// TIA Portal V17 export
// export: Created 2024-08-20T10:59:42.1994753Z, ExportSetting WithDefaults, DisplayName Totally Integrated Automation Portal, DisplayVersion V17 Update 4, DisplayName TIA Portal Openness, DisplayVersion V17 Update 4, DisplayName TIA Portal Version Control Interface, DisplayVersion V17, DisplayName STEP 7 Professional, DisplayVersion V17 Update 4, DisplayName STEP 7 Safety, DisplayVersion V17, DisplayName WinCC Advanced, DisplayVersion V17 Update 4
DATA_BLOCK "Digitais"   // DB300
{ S7_Optimized_Access := 'FALSE' }
VERSION : 0.1
// stored: AutoNumber false, DBAccessibleFromOPCUA true, IsOnlyStoredInLoadMemory false, IsWriteProtectedInAS false
   VAR RETAIN
      "MB-01-YSH" : Bool;   // Elevatoria principal 1 ligado
      "MB-01-YR" : Bool;   // Elevatoria principal 1 remoto
      "MB-01-YF" : Bool;   // Elevatoria principal 1 falha
      "MB-01-YFF" : Bool;   // Elevatoria principal 1 falta de fase
      "MB-01-MM" : Bool;   // Elevatoria principal 1 modo manutenção
      "MB-01-MA" : Bool;   // Elevatoria principal 1 modo automatico
      "MB-01-EMER" : Bool;   // Elevatoria principal 1 emergencia
      "MB-01-MN" : Bool;   // Elevatoria principal 1 modo normal
      "MB-01-ML" : Bool;   // Elevatoria principal 1 modo local
      "MB-01-YFI" : Bool;   // Elevatoria principal 1 com falha no inversor
      "MB-01-YFA" : Bool;   // Elevatoria principal 1 com falha no acionamento
      "MB-01-YPTA" : Bool;   // Elevatoria principal 1 com proteção térmica atuada
      "MB-01-HM" : Bool;   // Elevatoria principal 1 habilita manutenção
      "MB-01-RST" : Bool;   // Elevatoria principal 1 reset
      "MB-01-INTRU" : Bool;   // Elevatoria principal 1 intrusão no painel
      "MB-01-YFB" : Bool;   // Elevatoria principal 1 defeito na bomba
      "MB-02-YSH" : Bool;   // Elevatoria principal 2 ligado
      "MB-02-YR" : Bool;   // Elevatoria principal 2 remoto
      "MB-02-YF" : Bool;   // Elevatoria principal 2 falha
      "MB-02-YFF" : Bool;   // Elevatoria principal 2 falta de fase
      "MB-02-MM" : Bool;   // Elevatoria principal 2 modo manutenção
      "MB-02-MA" : Bool;   // Elevatoria principal 2 modo automatico
      "MB-02-EMER" : Bool;   // Elevatoria principal 2 emergencia
      "MB-02-MN" : Bool;   // Elevatoria principal 2 modo normal
      "MB-02-ML" : Bool;   // Elevatoria principal 2 modo local
      "MB-02-YFI" : Bool;   // Elevatoria principal 2 com falha no inversor
      "MB-02-YFA" : Bool;   // Elevatoria principal 2 com falha no acionamento
      "MB-02-YPTA" : Bool;   // Elevatoria principal 2 com proteção térmica atuada
      "MB-02-HM" : Bool;   // Elevatoria principal 2 habilita manutenção
      "MB-02-RST" : Bool;   // Elevatoria principal 2 reset
      "MB-02-INTRU" : Bool;   // Elevatoria principal 2 intrusão no painel
      "MB-02-YFB" : Bool;   // Elevatoria principal 2 defeito na bomba
      "MB-03-YSH" : Bool;   // Elevatoria principal 3 ligado
      "MB-03-YR" : Bool;   // Elevatoria principal 3 remoto
      "MB-03-YF" : Bool;   // Elevatoria principal 3 falha
      "MB-03-YFF" : Bool;   // Elevatoria principal 3 falta de fase
      "MB-03-MM" : Bool;   // Elevatoria principal 3 modo manutenção
      "MB-03-MA" : Bool;   // Elevatoria principal 3 modo automatico
      "MB-03-EMER" : Bool;   // Elevatoria principal 3 emergencia
      "MB-03-MN" : Bool;   // Elevatoria principal 3 modo normal
      "MB-03-ML" : Bool;   // Elevatoria principal 3 modo local
      "MB-03-YFI" : Bool;   // Elevatoria principal 3 com falha no inversor
      "MB-03-YFA" : Bool;   // Elevatoria principal 3 com falha no acionamento
      "MB-03-YPTA" : Bool;   // Elevatoria principal 3 com proteção térmica atuada
      "MB-03-HM" : Bool;   // Elevatoria principal 3 habilita manutenção
      "MB-03-RST" : Bool;   // Elevatoria principal 3 reset
      "MB-03-INTRU" : Bool;   // Elevatoria principal 3 intrusão no painel
      "MB-03-YFB" : Bool;   // Elevatoria principal 3 defeito na bomba
      "MB-04-YSH" : Bool;   // Elevatoria principal 4 ligado
      "MB-04-YR" : Bool;   // Elevatoria principal 4 remoto
      "MB-04-YF" : Bool;   // Elevatoria principal 4 falha
      "MB-04-YFF" : Bool;   // Elevatoria principal 4 falta de fase
      "MB-04-MM" : Bool;   // Elevatoria principal 4 modo manutenção
      "MB-04-MA" : Bool;   // Elevatoria principal 4 modo automatico
      "MB-04-EMER" : Bool;   // Elevatoria principal 4 emergencia
      "MB-04-MN" : Bool;   // Elevatoria principal 4 modo normal
      "MB-04-ML" : Bool;   // Elevatoria principal 4 modo local
      "MB-04-YFI" : Bool;   // Elevatoria principal 4 com falha no inversor
      "MB-04-YFA" : Bool;   // Elevatoria principal 4 com falha no acionamento
      "MB-04-YPTA" : Bool;   // Elevatoria principal 4 com proteção térmica atuada
      "MB-04-HM" : Bool;   // Elevatoria principal 4 habilita manutenção
      "MB-04-RST" : Bool;   // Elevatoria principal 4 reset
      "MB-04-INTRU" : Bool;   // Elevatoria principal 4 intrusão no painel
      "MB-04-YFB" : Bool;   // Elevatoria principal 4 defeito na bomba
      "LIT_001-AL8" : Bool;   // Disponível para alarme
      "LIT_001-AL9" : Bool;   // Disponível para alarme
      "LIT_001-AL10" : Bool;   // Disponível para alarme
      "LIT_001-AL11" : Bool;   // Disponível para alarme
      "LIT_001-AL12" : Bool;   // Disponível para alarme
      "LIT_001-AL13" : Bool;   // Disponível para alarme
      "LIT_001-AL14" : Bool;   // Disponível para alarme
      "LIT_001-AL15" : Bool;   // Disponível para alarme
      "LIT_001-YHH" : Bool;   // Alarme de nível muito alto do tanque
      "LIT_001-YH" : Bool;   // Alarme de nível alto do tanque
      "LIT_001-YL" : Bool;   // Alarme de nível baixo do tanque
      "LIT_001-YLL" : Bool;   // Alarme de nível muito baixo do tanque
      "LIT_001-YFS" : Bool;   // Transmissor de nível do tanque com falha de sinal
      "LIT_001-AL5" : Bool;   // Disponível para alarme
      "LIT_001-AL6" : Bool;   // Disponível para alarme
      "LIT_001-AL7" : Bool;   // Disponível para alarme
      PCM_EEE_EMER : Bool;   // PCM-E-CF-01-04 BOTAO DE EMERGENCIA - ATUADO
      PCM_EEE_K27 : Bool;   // PCM-E-CF-01-04 RELE DE PROTECAO FUNCAO 27 - ATUADO
      PCM_EEE_DISJ_LIG : Bool;   // PCM-E-CF-01-04 DISJUNTOR GERAL STATUS - LIGADO
      PCM_EEE_DISJ_DESLIG : Bool;   // PCM-E-CF-01-04 DISJUNTOR GERAL STATUS - DESLIGADO
      PCM_EEE_DISJ_YFAL : Bool;   // PCM-E-CF-01-04 DISJUNTOR GERAL STATUS - FALHA
      PCM_EEE_DISJ_FAL_GR : Bool;   // PCM-E-CF-01-04 FALHA GERAL ATUADO
      PCM_EEE_TR01_KA3 : Bool;   // PCM-E-CF-01-04 TRANSFORMADOR -TR-01 ALARME TEMP 150°
      PCM_EEE_TR01_KA4 : Bool;   // PCM-E-CF-01-04 TRANSFORMADOR -TR-01 ALARME TEMP 155°
      PCM_EEE_TR01_KA5 : Bool;   // PCM-E-CF-01-04 TRANSFORMADOR -TR-01 FALHA PROTECAO
      PCM_EEE_INTRU : Bool;   // PCM-E-CF-01-04 INTRUSAO NO PAINEL (COLUNA 01~04)
      PCM_EEE_RSERVA_0 : Bool;   // PCM-E-CF-01-04 BIT RESERVA DA WORD
      PCM_EEE_RSERVA_1 : Bool;   // PCM-E-CF-01-04 BIT RESERVA DA WORD
      PCM_EEE_RSERVA_2 : Bool;   // PCM-E-CF-01-04 BIT RESERVA DA WORD
      PCM_EEE_RSERVA_3 : Bool;   // PCM-E-CF-01-04 BIT RESERVA DA WORD
      PCM_EEE_RSERVA_4 : Bool;   // PCM-E-CF-01-04 BIT RESERVA DA WORD
      PCM_EEE_RSERVA_5 : Bool;   // PCM-E-CF-01-04 BIT RESERVA DA WORD
      QGBT_EMER : Bool;   // QGBT-AUX-01 BOTAO DE EMERGENCIA ATUADO
      QGBT_K27 : Bool;   // QGBT-AUX-01 RELE DE PROTECAO FUNCAO 27/59 ATUADO
      QGBT_DJL : Bool;   // QGBT-AUX-01 DISJUNTOR GERAL STATUS - LIGADO
      QGBT_DJD : Bool;   // QGBT-AUX-01 DISJUNTOR GERAL STATUS - DESLIGADO
      QGBT_DJYFAL : Bool;   // QGBT-AUX-01 DISJUNTOR GERAL FALHA - TRIP
      QGBT_INTRU : Bool;   // QGBT-AUX-01 INTRUSAO NO PAINEL
      QGBT_RESERVA_0 : Bool;   // QGBT-AUX-01 BIT RESERVA DA WORD
      QGBT_RESERVA_1 : Bool;   // QGBT-AUX-01 BIT RESERVA DA WORD
      QGBT_RESERVA_2 : Bool;   // QGBT-AUX-01 BIT RESERVA DA WORD
      QGBT_RESERVA_3 : Bool;   // QGBT-AUX-01 BIT RESERVA DA WORD
      QGBT_RESERVA_4 : Bool;   // QGBT-AUX-01 BIT RESERVA DA WORD
      QGBT_RESERVA_5 : Bool;   // QGBT-AUX-01 BIT RESERVA DA WORD
      QGBT_RESERVA_6 : Bool;   // QGBT-AUX-01 BIT RESERVA DA WORD
      QGBT_RESERVA_7 : Bool;   // QGBT-AUX-01 BIT RESERVA DA WORD
      QGBT_RESERVA_8 : Bool;   // QGBT-AUX-01 BIT RESERVA DA WORD
      QGBT_RESERVA_9 : Bool;   // QGBT-AUX-01 BIT RESERVA DA WORD
      LSL_001 : Bool;   // CHAVE DE NIVEL -LSL-001
      LSH_001 : Bool;   // CHAVE DE NIVEL -LSH-001
      LSL_002 : Bool;   // CHAVE DE NIVEL -LSL-002
      LSH_002 : Bool;   // CHAVE DE NIVEL -LSH-002
      LS_RESERVA_0 : Bool;   // CHAVE DE NIVEL - LS BIT RESERVA DA WORD
      LS_RESERVA_1 : Bool;   // CHAVE DE NIVEL - LS BIT RESERVA DA WORD
      LS_RESERVA_2 : Bool;   // CHAVE DE NIVEL - LS BIT RESERVA DA WORD
      LS_RESERVA_3 : Bool;   // CHAVE DE NIVEL - LS BIT RESERVA DA WORD
      LS_RESERVA_4 : Bool;   // CHAVE DE NIVEL - LS BIT RESERVA DA WORD
      LS_RESERVA_5 : Bool;   // CHAVE DE NIVEL - LS BIT RESERVA DA WORD
      LS_RESERVA_6 : Bool;   // CHAVE DE NIVEL - LS BIT RESERVA DA WORD
      LS_RESERVA_7 : Bool;   // CHAVE DE NIVEL - LS BIT RESERVA DA WORD
      LS_RESERVA_8 : Bool;   // CHAVE DE NIVEL - LS BIT RESERVA DA WORD
      LS_RESERVA_9 : Bool;   // CHAVE DE NIVEL - LS BIT RESERVA DA WORD
      LS_RESERVA_10 : Bool;   // CHAVE DE NIVEL - LS BIT RESERVA DA WORD
      LS_RESERVA_11 : Bool;   // CHAVE DE NIVEL - LS BIT RESERVA DA WORD
      PCE_EEE_INTRU : Bool;   // INTRUSAO NO PAINEL
      PCE_EEE_UPS_ALM : Bool;   // UPS EM ALARME FALHA NA BATERIA
      PCE_EEE_UPS_FE : Bool;   // UPS EM OPERACAO FALTA DE ENERGIA
      PCE_EEE_UPS_CHAR : Bool;   // UPS EM ALARME BATERIA CARREGADA
      "PCM-E-CF-01-P100-YFC" : Bool;   // Falha de comunicação com medidor do PCM-E-CF-01
      "QGBT-AUX-01-P100-YFC" : Bool;   // Falha de comunicação com medidor do PCM-E-CF-02
   END_VAR
BEGIN
END_DATA_BLOCK
